Fanuc KAREL source: ko00088.KL

PROGRAM KO00088
%STACKSIZE=65535
%PRIORITY=65535
%NOLOCKGROUP
VAR
P1 : JOINTPOS9
P2 : XYZWPR
F : BOOLEAN
OUT : JOINTPOS9
BEGIN
F=TRUE
-- UNSAFE_SOURCE_IR line 11: CALL_RESULT MIRROR(convert_jointpos9_to_xyzwprext(P1), convert_xyzwpr_to_position(P2), F)
END KO00088
